FUNCTION_BLOCK Pusher (* Composite Function Block Type *)
  (* Standard: 61499-2 *)
  (* Version 0.0, 7/14/2016, Andrei, nxtControl GmbH, template *)
  PACKAGE Main;
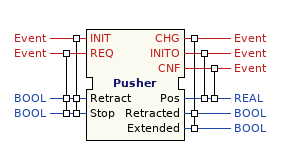
  EVENT_INPUT
    INIT WITH Retract, Stop; (* Initialization Request *)
    REQ WITH Retract, Stop; (* Normal Execution Request *)
  END_EVENT
  EVENT_OUTPUT
    CHG WITH Retracted, Extended;
    INITO WITH Pos; (* Initialization Confirm *)
    CNF WITH Pos; (* Execution Confirmation *)
  END_EVENT
  VAR_INPUT
    Retract : BOOL; (* Input event qualifier *)
    Stop : BOOL;
  END_VAR
  VAR_OUTPUT
    Pos : REAL; (* Output event qualifier *)
    Retracted : BOOL;
    Extended : BOOL;
  END_VAR
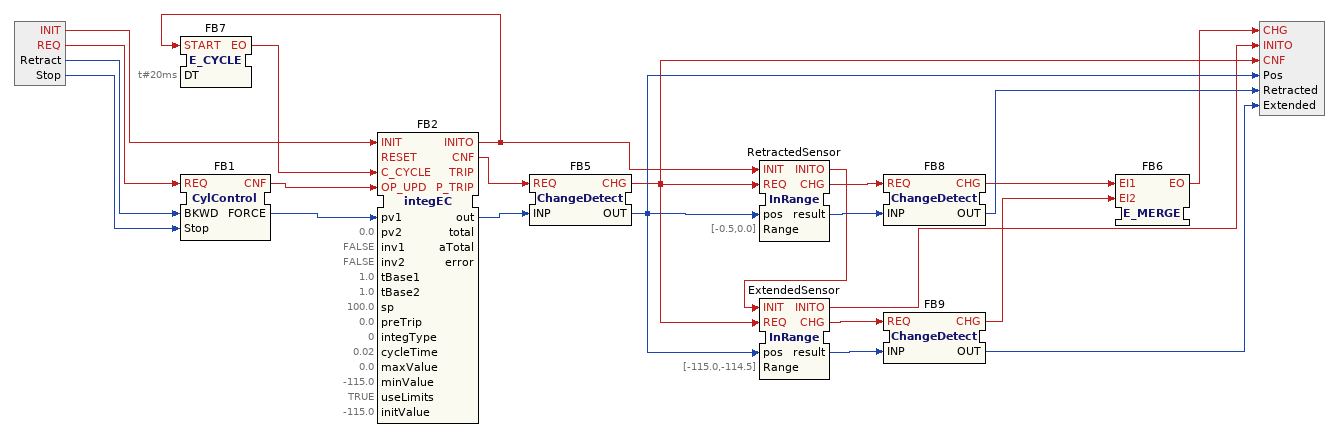
  FBS
    RetractedSensor : InRange(Range := [-0.5,0.0]);
    ExtendedSensor : InRange(Range := [-115.0,-114.5]);
    FB5 : ChangeDetect;
    FB6 : E_MERGE;
    FB7 : E_CYCLE(DT := t#20ms);
    FB8 : ChangeDetect;
    FB9 : ChangeDetect;
    FB1 : CylControl;
    FB2 : integEC(pv2 := 0.0, inv1 := FALSE, inv2 := FALSE, tBase1 := 1.0, tBase2 := 1.0, sp := 100.0, preTrip := 0.0, integType := 0, cycleTime := 0.02, maxValue := 0.0, minValue := -115.0, useLimits := TRUE, initValue := -115.0);
  END_FBS
  EVENT_CONNECTIONS
    FB1.CNF TO FB2.OP_UPD;
    FB2.CNF TO FB5.REQ;
    FB5.CHG TO RetractedSensor.REQ;
    FB5.CHG TO ExtendedSensor.REQ;
    FB2.INITO TO RetractedSensor.INIT;
    RetractedSensor.INITO TO ExtendedSensor.INIT;
    ExtendedSensor.INITO TO INITO;
    FB6.EO TO CHG;
    FB5.CHG TO CNF;
    FB7.EO TO FB2.C_CYCLE;
    INIT TO FB2.INIT;
    FB2.INITO TO FB7.START;
    REQ TO FB1.REQ;
    RetractedSensor.CHG TO FB8.REQ;
    ExtendedSensor.CHG TO FB9.REQ;
    FB8.CHG TO FB6.EI1;
    FB9.CHG TO FB6.EI2;
  END_CONNECTIONS
  DATA_CONNECTIONS
    FB1.FORCE TO FB2.pv1;
    FB2.out TO FB5.INP;
    FB5.OUT TO Pos;
    FB5.OUT TO ExtendedSensor.pos;
    FB5.OUT TO RetractedSensor.pos;
    Retract TO FB1.BKWD;
    Stop TO FB1.Stop;
    RetractedSensor.result TO FB8.INP;
    ExtendedSensor.result TO FB9.INP;
    FB8.OUT TO Retracted;
    FB9.OUT TO Extended;
  END_CONNECTIONS
END_FUNCTION_BLOCK
